FUNCTION_BLOCK FB_ManualControl
VAR_INPUT
END_VAR
VAR_OUTPUT
	fVelocityFeedForwardControlOutput : LREAL;
END_VAR
VAR
	fNormalizedJoystickY : LREAL;
	fbOpenLoopControl : FB_OpenLoopControl; 
	bEnable : BOOL := TRUE;
END_VAR

CASE Parameters.eErrorModes OF
	E_ErrorModes.MaxLimit:
		IF Inputs.fJoystickY > 0.0 THEN
			Inputs.fJoystickY := 0.0;
		END_IF
	E_ErrorModes.MinLimit:
		IF Inputs.fJoystickY < 0.0 THEN
			Inputs.fJoystickY := 0.0;
		END_IF
END_CASE 

fNormalizedJoystickY := Inputs.fJoystickY*Parameters.stCraneParameters.fMaxVelocityLimit;

fbOpenLoopControl(
	bEnable := bEnable,
	stParam := Parameters.stCraneParameters,
	fInput_ms := fNormalizedJoystickY,
	fMaxValveFlow_lmin := Parameters.stCraneParameters.fMaxFlowCapacity,
	fNormalizedOutput => Outputs.fNormalizedOutput
);

HMI.fCylinderPositon := Outputs.fNormalizedOutput;

END_FUNCTION_BLOCK

(* stored: Version 1.1.0.1, ProductVersion 3.1.4024.10
   POU FB_ManualControl: Id {ca9c3dcf-0c0f-42e0-a37d-836583731b5d}, SpecialFunc None *)
